(*
version 1.3	21. oct. 2008
programmer 	hugo
tested by	tobias

find_char searches str and returns the starting position of the first character that is not a control character.
control characters are the ascii character 00 .. 31 and 127

*)
FUNCTION FIND_CHAR : INT
VAR_INPUT
	str : STRING(STRING_LENGTH);
	pos : INT;
END_VAR
VAR
	i: INT;
	pt : POINTER TO ARRAY[1..255] OF BYTE;
	stop: INT;
	X: BYTE;
END_VAR

pt := ADR(str);
stop := LEN(str);
FOR i := MAX(pos,1) TO stop DO;
	X := pt^[i];
	IF X > 31 AND ((setup.EXTENDED_ASCII AND X <> 127) OR (NOT setup.EXTENDED_ASCII AND X < 127)) THEN
		FIND_CHAR := i;
		RETURN;
	END_IF;
END_FOR;
FIND_CHAR := 0;


(* revision history
hm	29. feb 2008	rev 1.0
	original version

hm	26. mar. 2008	rev 1.1
	char will now accept extended ascii

hm	29. mar. 2008	rev 1.2
	changed STRING to STRING(STRING_LENGTH)

hm	21. oct. 2008	rev 1.3
	changes setup constants
	optimized code
*)

END_FUNCTION

(* stored: Version 1.1.0.1
   POU FIND_CHAR: Id {4414ee9f-f75a-4f62-b396-9b9952c84e5a}, SpecialFunc None *)
